(* CODESYS project HTTPSClient.library
   LanguageModelAttribute: qualified-access-only
   DefaultNamespace: HTTPS
   Description: HTTPS Client for sending http request to a webserver.
   Author: Turck Vilant Oy
   DocFormat: reStructuredText
   Title: HTTPS Client
   Version: 1.0.0.1
   Company: CODESYS GmbH
   Placeholder: HTTPSClient

Project tree, tasks and I/O mapping:
  libraries: CAA Behaviour Model, 3.5.19.0 (CAA Technical Workgroup); StringUtils, 3.5.18.0 (System); Util, 3.5.19.0 (System); Net Base Services, 3.5.19.20 (3S - Smart Software Solutions GmbH)
  HTTPRequest/
    Function Blocks/
      function block HttpsClient [ST]: StartAction, StringToURL, CyclicAction, prvResetOutputs, CreateRequest, ResetAction, prvAbort, ParseResult
    Enums/
      data type STATE
      data type REQUEST_TYPE
      data type ERROR
      data type CONTENT_TYPE
    Structs/
      data type URL
      data type HttpResult
    Functions/
      function URLDecoder [ST]
      BASE64/
        function block BASE64_DECODE [ST]
        function block BASE64_ENCODE [ST]
        function CODE [ST]
      UTF-8/
        global variables GVL_UTF8
        function ConvertUTF16toUTF8 [ST]
        function ConvertUTF8toUTF16 [ST]
        function IsLegalUTF8 [ST]
      function Concat [ST]
    Constants/
      global variables GVL
    Params/
      global variables Param
  00000000-0000-0000-0000-000000000000|C:\Users\m.lamp\Documents\license.txt
  license
*)

// HTTPRequest/Enums/STATE
// State of requests
{attribute 'qualified_only'}
{attribute 'hide'}
TYPE STATE :
(
	START := 0,
	INIT,
	REQUEST,
	RESPONSE,
	ERROR,
	IDLE
);
END_TYPE

// HTTPRequest/Enums/REQUEST_TYPE
// Types of http requests
TYPE REQUEST_TYPE :
(
	GET := 0, // http GET
	POST := 1, // http POST (needs input pwsPostValue) 
	DELETE := 2, // http DELETE
	PUT := 3, // http PUT (needs input pwsPostValue) 
	HEAD := 4 // http HEAD
);
END_TYPE

// HTTPRequest/Structs/URL
// URL structure
TYPE URL :
STRUCT
	wsProtocol	: WSTRING(5); 	// Protocol e.g. http, NOTE: ONLY HTTP IS SUPPORTED! 
	wsDomain	: WSTRING(255); 	// The domain e.g. 'twitter.api.com'
	uiPort		: UINT;			// Port of the server
	wsPath		: WSTRING(255);	// The path e.g. '/1.1/statuses/update.json'
END_STRUCT
END_TYPE

// HTTPRequest/Enums/ERROR
{attribute 'qualified_only'}
TYPE ERROR :
(
	NO_ERROR := 0, // No error
	TIME_OUT := 1, // Time out
	UNEXPECTED_ERROR := 2, // Unexpected error
	TCP_INIT_ERROR := 3, // Unable to initialize the TCP socket
	TCP_READ_ERROR := 4, // Error while reading response
	TCP_WRITE_ERROR := 5, // Error while sending the request
	MISSING_POST_VALUE := 6, // Current request type needs a post value
	RESULT_PARSE_ERROR := 7 // Error while parsing the response
);
END_TYPE

// HTTPRequest/Structs/HttpResult
// The result of a http request
TYPE HttpResult :
STRUCT
	iStatus					: INT; // http status
	wsHeader				: WSTRING(g_udiMaxHeaderSize); // http header as WSTRING
	wsContent				: WSTRING(g_udiMaxResponseSize); // The result of the request as WSTRING
	sHeader					: STRING(g_udiMaxHeaderSize); // http header as STRING
	sContent				: STRING(g_udiMaxResponseSize); // The result of the request as STRING
	diContentLength			: DINT; // Length of wsContent
END_STRUCT
END_TYPE

// HTTPRequest/Enums/CONTENT_TYPE
{attribute 'qualified_only'}
{attribute 'strict'}
TYPE CONTENT_TYPE :
(
	APPLICATION_FORM := 0, // HTML-Formulardaten an CGI 
	APPLICATION_JSON // enthält einen String in JavaScript-Objekt-Notation
);
END_TYPE

// HTTPRequest/Constants/GVL
{attribute 'hide'}
VAR_GLOBAL CONSTANT
	gc_wsBLANK : WSTRING(1) := " ";
	gc_wsLF	: WSTRING(2) :=	"$R$N";
	gc_wsDoubleLF	: WSTRING(4) :=	"$R$N$R$N";
	gc_wsContentLength	: WSTRING(15) := "Content-Length:";
	gc_wsChunked		: WSTRING(26) := "Transfer-Encoding: chunked";
	gc_wsHex	: WSTRING(3) :=	"16#";
END_VAR

// HTTPRequest/Functions/UTF-8/GVL_UTF8
{attribute 'hide'}
VAR_GLOBAL CONSTANT
	trailingBytesForUTF8 : ARRAY[0..255] OF BYTE := [
				0,0,0,0,0,0,0,0,0,0,0,0,0,0,0,0, 0,0,0,0,0,0,0,0,0,0,0,0,0,0,0,0,
				0,0,0,0,0,0,0,0,0,0,0,0,0,0,0,0, 0,0,0,0,0,0,0,0,0,0,0,0,0,0,0,0,
				0,0,0,0,0,0,0,0,0,0,0,0,0,0,0,0, 0,0,0,0,0,0,0,0,0,0,0,0,0,0,0,0,
				0,0,0,0,0,0,0,0,0,0,0,0,0,0,0,0, 0,0,0,0,0,0,0,0,0,0,0,0,0,0,0,0,
				0,0,0,0,0,0,0,0,0,0,0,0,0,0,0,0, 0,0,0,0,0,0,0,0,0,0,0,0,0,0,0,0,
				0,0,0,0,0,0,0,0,0,0,0,0,0,0,0,0, 0,0,0,0,0,0,0,0,0,0,0,0,0,0,0,0,
				1,1,1,1,1,1,1,1,1,1,1,1,1,1,1,1, 1,1,1,1,1,1,1,1,1,1,1,1,1,1,1,1,
				2,2,2,2,2,2,2,2,2,2,2,2,2,2,2,2, 3,3,3,3,3,3,3,3,4,4,4,4,5,5,5,5
			];
	firstByteMark : ARRAY[0..6] OF BYTE := [ 16#00, 16#00, 16#C0, 16#E0, 16#F0, 16#F8, 16#FC ];
	
	offsetsFromUTF8: ARRAY[0..5] OF DWORD := [ 16#00000000, 16#00003080, 16#000E2080, 
             16#03C82080, 16#FA082080, 16#82082080 ];
	
	halfShift : INT := 10; (* used FOR shifting BY 10 bits *)

	halfBase : DWORD := 16#0010000;
	halfMask : DWORD := 16#3FF;
	
	UNI_REPLACEMENT_CHAR : DWORD := 16#0000FFFD;
	
	UNI_MAX_BMP : DWORD := 16#0000FFFF;
	UNI_MAX_UTF16 : DWORD := 16#0010FFFF;
	UNI_MAX_UTF32 : DWORD := 16#7FFFFFFF;
	UNI_MAX_LEGAL_UTF32 : DWORD := 16#0010FFFF;
	
	byteMask : DWORD := 16#BF;
	byteMark : DWORD := 16#80;
	UNI_SUR_HIGH_START : DWORD := 16#D800;
 	UNI_SUR_HIGH_END : DWORD := 16#DBFF;
 	UNI_SUR_LOW_START : DWORD := 16#DC00;
 	UNI_SUR_LOW_END : DWORD := 16#DFFF;
	
	ERR_OK : UDINT := 16#0000;	(* The operation succeeded *)
	ERR_SOURCE_EXHAUSTED : UDINT := 16#40A0; (* Used for UTF8 helper *)
	ERR_TARGET_EXHAUSTED : UDINT := 16#40A1; (* Used for UTF8 helper *)
	ERR_SOURCE_ILLEGAL : UDINT := 16#40A2; (* Used for UTF8 helper *)
	
END_VAR

// HTTPRequest/Params/Param
// HTTPClient parameters
VAR_GLOBAL CONSTANT
	g_udiMaxRequestSize : UDINT := 16000; // Maximum size of the http request in btyes
	g_udiMaxResponseSize : UDINT := 16000; // Maximum size of the http response in bytes
	g_udiMaxHeaderSize : UDINT := 4000; // Maximum size of the http header in bytes
END_VAR

// HTTPRequest/Function Blocks/HttpsClient
// Functionblock to send http GET and POST requests.
//{attribute 'hide_all_locals'}
FUNCTION_BLOCK HttpsClient EXTENDS CBM.ETrigTo
VAR_INPUT
	sURL					: STRING(1024); // URL of the web server
	eRequestType			: REQUEST_TYPE := REQUEST_TYPE.GET;	// Type of the request: POST or GET
	eContentType			: CONTENT_TYPE := CONTENT_TYPE.APPLICATION_FORM; // HTTP Content-Type of the request
	pwsAdditionalHeader		: POINTER TO WSTRING; // Additional HTTP header
	pwsPostValue			: POINTER TO WSTRING; // Post parameter
	httpsTLSContext 		: NBS.ITLSContext := 0; // TLS context for HTTPS
END_VAR
VAR_OUTPUT
	eError					: ERROR; // Current error state
	httpResult				: HttpResult; // The result of the request
	_url					: URL;
	// Helpers	
	_eState 				: STATE;
END_VAR
VAR
	// TCP Connection
	_tcp_client 			: NBS.TCP_Client;
	_tcp_read 				: NBS.TCP_Read;
	_tcp_write 				: NBS.TCP_Write;
	_IPAddr 				: NBS.IPv4Address := (ipAddress := '83.150.96.4');
	_IIPAddr	 			: NBS.IIPAddress := _IPAddr;
	_resolve_host_name 		: NBS.ResolveHostname;	
	_wsRequest 				: WSTRING(g_udiMaxRequestSize);
	_abRequest 				: ARRAY[0..g_udiMaxRequestSize] OF BYTE;
	_sContent				: STRING(g_udiMaxResponseSize); 
	_pbContent				: POINTER TO BYTE;
	_wsContent				: WSTRING(g_udiMaxResponseSize);
	
	
END_VAR

SUPER^();
eError := iError;

{attribute 'hide'}
METHOD StartAction : BOOL
VAR_INPUT
END_VAR
VAR
END_VAR
END_METHOD

{attribute 'hide'}
// Converts a string to an url.
METHOD StringToURL : ERROR
VAR_INPUT
	wsUrl		: WSTRING(1024);	// The url as string
END_VAR
VAR_IN_OUT
	url			: URL; // The URL struct
END_VAR
VAR
	wsTemp		: WSTRING(1024);
	wsPort		: WSTRING(6);
	i			: INT;
END_VAR
VAR CONSTANT
	wsDel		: WSTRING(3) := "://";
	wsPortDel	: WSTRING(1) := ":";
	wsPathStart	: WSTRING(1) := "/";
END_VAR
// Find '://'
i := Stu.StrFindW(pst1 := ADR(wsUrl), pst2 := ADR(wsDel), uiSearchStart := 1);
IF i > 0 THEN
	Stu.StrMidW(pwst := ADR(wsUrl),
				uiInputBufferSize := SIZEOF(wsUrl),
				iLength := DINT_TO_INT(Stu.StrLenW(ADR(wsUrl))) - i - DINT_TO_INT(Stu.StrLenW(ADR(wsDel))) + 1,
				iPosition := i +  DINT_TO_INT(Stu.StrLenW(ADR(wsDel))),
				pwstResult := ADR(wsTemp),
				uiResultBufferSize := SIZEOF(wsTemp));
	// Set protocol			
	Stu.StrMidW(pwst := ADR(wsUrl),
				uiInputBufferSize := SIZEOF(wsUrl),
				iLength := i - 1,
				iPosition := 1,
				pwstResult := ADR(url.wsProtocol),
				uiResultBufferSize := SIZEOF(url.wsProtocol));
ELSE
	url.wsProtocol := "http";
	wsTemp := wsUrl;
END_IF

// Find path start '/'
i := Stu.StrFindW(pst1 := ADR(wsTemp), pst2 := ADR(wsPathStart), uiSearchStart := 1);
IF i > 0 THEN
	// set path
	Stu.StrMidW(pwst := ADR(wsTemp),
				uiInputBufferSize := SIZEOF(wsTemp),
				iLength := DINT_TO_INT(Stu.StrLenW(ADR(wsTemp))) - i + DINT_TO_INT(Stu.StrLenW(ADR(wsPathStart))),
				iPosition := i + DINT_TO_INT(Stu.StrLenW(ADR(wsPathStart))) - 1,
				pwstResult := ADR(url.wsPath),
				uiResultBufferSize := SIZEOF(url.wsPath));	
				
	Stu.StrMidW(pwst := ADR(wsTemp),
				uiInputBufferSize := SIZEOF(wsTemp),
				iLength := i - 1,
				iPosition := 1,
				pwstResult := ADR(wsTemp),
				uiResultBufferSize := SIZEOF(wsTemp));			
ELSE
	url.wsPath := "";
END_IF


i := Stu.StrFindW(pst1 := ADR(wsTemp), pst2 := ADR(wsPortDel), uiSearchStart := 1);
IF i > 0 THEN
	// set domain
	Stu.StrMidW(pwst := ADR(wsTemp),
				uiInputBufferSize := SIZEOF(wsTemp),
				iLength := i - 1,
				iPosition := 1,
				pwstResult := ADR(url.wsDomain),
				uiResultBufferSize := SIZEOF(url.wsDomain));	
	// set port
	Stu.StrMidW(pwst := ADR(wsTemp),
				uiInputBufferSize := SIZEOF(wsTemp),
				iLength := DINT_TO_INT(Stu.StrLenW(ADR(wsTemp)) - i - Stu.StrLenW(ADR(wsPortDel))) + 1,
				iPosition := i + DINT_TO_INT(Stu.StrLenW(ADR(wsPortDel))),
				pwstResult := ADR(wsPort),
				uiResultBufferSize := SIZEOF(wsPort));
	url.uiPort := WSTRING_TO_UINT(wsPort);				
ELSIF url.wsProtocol = "http" THEN
	url.wsDomain := wsTemp;
	url.uiPort := 80;
ELSIF url.wsProtocol = "https" THEN
	url.wsDomain := wsTemp;
	url.uiPort := 443;
ELSE
	url.wsDomain := wsTemp;
	url.uiPort := 80;
END_IF

IF url.wsPath = "" THEN
	url.wsPath := "/";
END_IF
END_METHOD

{attribute 'hide'}
METHOD CyclicAction : BOOL
VAR_INPUT
END_VAR
VAR
	uxiBytesRead : __UXINT;
	sDomain : STRING;
END_VAR

IF xExecute = TRUE AND _eState = STATE.IDLE THEN
	_eState := STATE.START;
END_IF

CASE _eState OF
	
STATE.IDLE: // Idle

STATE.START: // stopped
	// Parse url 
	_sContent := '';
	_pbContent := ADR(_sContent);
	_wsContent := "";
	httpResult.wsContent := "";
	httpResult.wsHeader := "";
	httpResult.diContentLength := 0;
	httpResult.iStatus := 0;
	iError := StringToURL(wsUrl := STRING_TO_WSTRING(sUrl), url := _url);
	IF iError <> ERROR.NO_ERROR THEN
		_eState := STATE.ERROR;		
		xError := TRUE;	
		RETURN;
	END_IF
	//_IPAddr.sAddr := WSTRING_TO_STRING(_url.wsDomain);
	_tcp_client(xEnable := FALSE);
	_tcp_read(xEnable := FALSE);
	_tcp_write(xExecute := FALSE);
	sDomain := WSTRING_TO_STRING(_url.wsDomain);
	_resolve_host_name(xExecute:=, sHostName:=sDomain , itfIPAddress:=_IIPAddr);
	_resolve_host_name.xExecute := TRUE;
	IF _resolve_host_name.xDone THEN
		_resolve_host_name.xExecute := FALSE;
		_eState := STATE.INIT;
	END_IF
	
	IF (eRequestType = REQUEST_TYPE.POST OR eRequestType = REQUEST_TYPE.PUT) AND (pwsPostValue = 0 OR Stu.StrLenW(pstData := pwsPostValue) = 0) THEN
		iError := ERROR.MISSING_POST_VALUE;
		_eState := STATE.ERROR;
	END_IF
	
STATE.INIT:	// init client
	_tcp_client(xEnable := TRUE, itfIPAddress := _IIPAddr, uiPort := _url.uiPort, itfTLSContext:=httpsTLSContext);
	IF _tcp_client.xBusy THEN//AND _tcp_client.hConnection <> CAA.gc_hINVALID THEN
		_eState := STATE.REQUEST;
	ELSIF _tcp_client.xError THEN
		iError := ERROR.TCP_INIT_ERROR;
		_eState := STATE.ERROR;
	END_IF
	
STATE.REQUEST:		// send message	
	CreateRequest(url := _url, pwsAdditionalHeader := pwsAdditionalHeader, pwsPostValue := pwsPostValue, wsOut := _wsRequest);
	ConvertUTF16toUTF8(sourceStart := ADR(_wsRequest), targetStart := ADR(_abRequest), dwTargetBufferSize := SIZEOF(_abRequest), bStrictConversion := FALSE);
	_tcp_write(xExecute := _tcp_client.xActive, itfConnection := _tcp_client.itfConnection, udiSize := DINT_TO_UDINT(Stu.StrLenA(ADR(_abRequest))), pData := ADR(_abRequest));
	IF _tcp_write.xDone THEN		// message sent, go back to idle mode
		_tcp_write(xExecute := FALSE);			
		_eState := STATE.RESPONSE;
	ELSIF _tcp_write.xError THEN
		iError := ERROR.TCP_WRITE_ERROR;
		_eState := STATE.ERROR;
	END_IF
	
STATE.RESPONSE:	// idle mode - wait for incomming message
	_tcp_read(xEnable := _tcp_client.xActive, itfConnection := _tcp_client.itfConnection, udiSize := SIZEOF(_sContent), pData := ADR(_sContent));
	IF _tcp_read.xReady THEN		
		_pbContent[uxiBytesRead] := 0;
		_tcp_read(xEnable := FALSE);		
		_eState := STATE.IDLE;
		ResetAction();
		ConvertUTF8toUTF16(sourceStart := ADR(_sContent), targetStart := ADR(_wsContent), dwTargetBufferSize := SIZEOF(_wsContent), bStrictConversion := FALSE);
		ParseResult(wsContent := _wsContent, httpResult := httpResult);
		xDone := TRUE;
	ELSIF _tcp_read.xError THEN		
		iError := ERROR.TCP_READ_ERROR;
		_eState := STATE.ERROR;		
		xError := TRUE;	
	END_IF		

STATE.ERROR:
	_sContent := '';
	_wsContent := "";
	ResetAction();
	_eState := STATE.IDLE;
	
END_CASE
END_METHOD

{attribute 'hide'}
METHOD prvResetOutputs : BOOL
VAR_INPUT
END_VAR
VAR
END_VAR
SUPER^.prvResetOutputs();
END_METHOD

// Builds a http request
{attribute 'hide'}
METHOD CreateRequest
VAR_INPUT
	url						: URL; // The URL of the webserver
	pwsAdditionalHeader		: POINTER TO WSTRING; // Additional HTTP header	
	pwsPostValue			: POINTER TO WSTRING; // Post parameter
END_VAR
VAR_IN_OUT
	wsOut					: WSTRING(g_udiMaxRequestSize);
END_VAR
VAR
	wsType				: WSTRING(6); // Type of the request: GET or POST
	wsContentLength		: WSTRING(5);
	wsHTTP_HEADER		: WSTRING(100) 	:= "Connection: close$000D$000AContent-Type: application/x-www-form-urlencoded";
END_VAR
VAR CONSTANT
	wsBlank				: WSTRING(1) 	:= " ";
	wsLF				: WSTRING(2) 	:= "$000D$000A";
	wsLF2				: WSTRING(4) 	:= "$000D$000A$000D$000A";
	wsHTTPVersion		: WSTRING(12) 	:= " HTTP/1.1";
	wsHTTPContetntLength	: WSTRING(17) 	:= "Content-Length: ";
	wsHTTPHost 			: WSTRING(9) 	:= "Host: ";
END_VAR
IF eRequestType = REQUEST_TYPE.GET THEN
	wsType := "GET";
ELSIF eRequestType = REQUEST_TYPE.DELETE THEN
	wsType := "DELETE";
ELSIF eRequestType = REQUEST_TYPE.HEAD THEN
	wsType := "HEAD";
ELSIF eRequestType = REQUEST_TYPE.PUT THEN
	wsType := "PUT";
ELSIF eRequestType = REQUEST_TYPE.POST THEN
	wsType := "POST";
ELSE
	wsType := "";
END_IF

IF eContentType = CONTENT_TYPE.APPLICATION_JSON THEN
	wsHTTP_HEADER := "Connection: keep-alive$000D$000AContent-Type: application/json";
END_IF

// POST or GET
wsOut := "";
Concat(ADR(wsType), ADR(wsOut), SIZEOF(wsOut));
Concat(ADR(wsBlank), ADR(wsOut), SIZEOF(wsOut));
Concat(ADR(url.wsPath), ADR(wsOut), SIZEOF(wsOut));
Concat(ADR(wsBlank), ADR(wsOut), SIZEOF(wsOut));
Concat(ADR(wsHTTPVersion), ADR(wsOut), SIZEOF(wsOut));
Concat(ADR(wsLF), ADR(wsOut), SIZEOF(wsOut));

// HTTP Header
Stu.StrConcatW(ADR(wsHTTP_HEADER), ADR(wsOut), DINT_TO_INT(SIZEOF(wsOut)));
Stu.StrConcatW(ADR(wsLF), ADR(wsOut), DINT_TO_INT(SIZEOF(wsOut)));
IF NOT Stu.StrIsNullOrEmptyA(pwsAdditionalHeader) THEN
	Stu.StrConcatW(pwsAdditionalHeader, ADR(wsOut), DINT_TO_INT(SIZEOF(wsOut)));
	Stu.StrConcatW(ADR(wsLF), ADR(wsOut), DINT_TO_INT(SIZEOF(wsOut)));
END_IF

// Host
Concat(ADR(wsHTTPHost), ADR(wsOut), SIZEOF(wsOut));
Concat(ADR(url.wsDomain), ADR(wsOut), SIZEOF(wsOut));
Concat(ADR(wsLF), ADR(wsOut), SIZEOF(wsOut));

IF eRequestType = REQUEST_TYPE.POST OR eRequestType = REQUEST_TYPE.PUT THEN
	Concat(ADR(wsHTTPContetntLength), ADR(wsOut), SIZEOF(wsOut));
	wsContentLength := DINT_TO_WSTRING(Stu.StrLenW(pwsPostValue));
	Concat(ADR(wsContentLength), ADR(wsOut), SIZEOF(wsOut));
END_IF
Concat(ADR(wsLF), ADR(wsOut), SIZEOF(wsOut));
Concat(ADR(wsLF), ADR(wsOut), SIZEOF(wsOut));

// Post content
IF eRequestType = REQUEST_TYPE.POST OR eRequestType = REQUEST_TYPE.PUT THEN
	Concat(pwsPostValue, ADR(wsOut), SIZEOF(wsOut));
END_IF
END_METHOD

{attribute 'hide'}
METHOD ResetAction
VAR_INPUT
END_VAR
_tcp_write(xExecute := FALSE);	
_tcp_read(xEnable := FALSE);	
_tcp_client(xEnable := FALSE);
END_METHOD

{attribute 'hide'}
METHOD prvAbort : BOOL
VAR_INPUT
END_VAR
VAR
END_VAR
ResetAction();
_eState := STATE.IDLE;
xAbortInProgress := FALSE;
END_METHOD

{attribute 'hide'}
METHOD ParseResult : ERROR
VAR_IN_OUT
	wsContent : WSTRING(g_udiMaxResponseSize);
	httpResult : HTTPResult;
END_VAR
VAR
	diTemp1 : DINT;
	diTemp2 : DINT;
	diContentStartPos : DINT;
	wsStatus : WSTRING(4);
	wsContentLength : WSTRING(20);
	wsContentLengthHex : WSTRING(20);
	xIsChunked : BOOL;
END_VAR
// Find HTTP status
diTemp1 := Stu.StrFindW(pst1 := ADR(wsContent), pst2 := ADR(gc_wsBLANK), uiSearchStart := 0);
diTemp2 := Stu.StrFindW(pst1 := ADR(wsContent), pst2 := ADR(gc_wsBLANK), uiSearchStart := DINT_TO_UINT(diTemp1 + 1));
IF diTemp1 < 1 OR diTemp2 < 1 THEN
	ParseResult := ERROR.RESULT_PARSE_ERROR;
	RETURN;
END_IF
Stu.StrMidW(	pwst := ADR(wsContent), 
				uiInputBufferSize := SIZEOF(wsContent), 
				iLength := DINT_TO_INT(diTemp2 - diTemp1), 
				iPosition := DINT_TO_INT(diTemp1), 
				pwstResult := ADR(wsStatus), 
				uiResultBufferSize := SIZEOF(wsStatus));
httpResult.iStatus := WSTRING_TO_INT(wsStatus);

// Find header
diTemp1 := Stu.StrFindW(pst1 := ADR(wsContent), pst2 := ADR(gc_wsLF), uiSearchStart := DINT_TO_UINT(diTemp2 + 1));
diTemp2 := Stu.StrFindW(pst1 := ADR(wsContent), pst2 := ADR(gc_wsDoubleLF), uiSearchStart := DINT_TO_UINT(diTemp1 + 1));
IF diTemp1 < 1 OR diTemp2 < 1 THEN
	ParseResult := ERROR.RESULT_PARSE_ERROR;
	RETURN;
END_IF
Stu.StrMidW(	pwst := ADR(wsContent), 
				uiInputBufferSize := SIZEOF(wsContent), 
				iLength := DINT_TO_INT(diTemp2 - diTemp1) - 2, 
				iPosition := DINT_TO_INT(diTemp1) + 2, 
				pwstResult := ADR(httpResult.wsHeader), 
				uiResultBufferSize := SIZEOF(httpResult.wsHeader));

diContentStartPos := diTemp2 + 4;

xIsChunked := Stu.StrFindW(pst1 := ADR(httpResult.wsHeader), pst2 := ADR(gc_wsChunked), uiSearchStart := 0) > 0;
IF xIsChunked THEN
	// Convert chunked data
	diTemp1 := diContentStartPos;
	// Get data length
	diTemp2 := Stu.StrFindW(pst1 := ADR(wsContent), pst2 := ADR(gc_wsLF), uiSearchStart := DINT_TO_UINT(diTemp1));
	IF diTemp2 < 1 THEN
		ParseResult := ERROR.RESULT_PARSE_ERROR;
		RETURN;
	END_IF
	Stu.StrMidW(	pwst := ADR(wsContent), 
					uiInputBufferSize := SIZEOF(wsContent), 
					iLength := DINT_TO_INT(diTemp2 - diTemp1), 
					iPosition := DINT_TO_INT(diTemp1), 
					pwstResult := ADR(wsContentLength), 
					uiResultBufferSize := SIZEOF(wsContentLength));
	wsContentLengthHex := gc_wsHex;
	Stu.StrConcatW(pstFrom := ADR(wsContentLength), pstTo := ADR(wsContentLengthHex), iBufferSize := SIZEOF(wsContentLengthHex));
	httpResult.diContentLength := WSTRING_TO_DINT(wsContentLengthHex);
	// Copy content
	Stu.StrMidW(	pwst := ADR(wsContent), 
					uiInputBufferSize := SIZEOF(wsContent), 
					iLength := DINT_TO_INT(httpResult.diContentLength), 
					iPosition := DINT_TO_INT(diTemp2 + 2), 
					pwstResult := ADR(httpResult.wsContent), 
					uiResultBufferSize := SIZEOF(httpResult.wsContent));
ELSE	
	// Find content
	diTemp2 := Stu.StrLenW(pstData := ADR(wsContent));
	IF diTemp2 < 0 THEN
		ParseResult := ERROR.RESULT_PARSE_ERROR;
		RETURN;
	END_IF
	Stu.StrMidW(	pwst := ADR(wsContent), 
					uiInputBufferSize := SIZEOF(wsContent), 
					iLength := DINT_TO_INT(diTemp2 - diContentStartPos + 1), 
					iPosition := DINT_TO_INT(diContentStartPos), 
					pwstResult := ADR(httpResult.wsContent), 
					uiResultBufferSize := SIZEOF(httpResult.wsContent));
	httpResult.diContentLength := diTemp2 - diContentStartPos + 1;
END_IF

// Copy WSTRING to STRING values
ConvertUTF16toUTF8(sourceStart := ADR(httpResult.wsHeader), targetStart := ADR(httpResult.sHeader), dwTargetBufferSize := SIZEOF(httpResult.sHeader), bStrictConversion := FALSE);
ConvertUTF16toUTF8(sourceStart := ADR(httpResult.wsContent), targetStart := ADR(httpResult.sContent), dwTargetBufferSize := SIZEOF(httpResult.sContent), bStrictConversion := FALSE);
END_METHOD

END_FUNCTION_BLOCK

// HTTPRequest/Functions/UTF-8/ConvertUTF16toUTF8
// Converts a WSTRING to STRING
FUNCTION ConvertUTF16toUTF8 : UDINT
VAR_INPUT
 	sourceStart : POINTER TO WORD;	// Pointer to WSTRING
	targetStart : POINTER TO BYTE;	// Pointer to STRING
	dwTargetBufferSize : DWORD;		// Size of STRING
	bStrictConversion : BOOL;
END_VAR
VAR
	source : POINTER TO WORD;
	sourceEnd : POINTER TO WORD;
	oldSource : POINTER TO WORD;
	target : POINTER TO BYTE;
	targetEnd : POINTER TO BYTE;
	ch : DWORD;
	ch2 : DWORD;
	bytesToWrite : WORD := 0;
	bytesToWriteSave : WORD := 0;
END_VAR

ConvertUTF16toUTF8 := ERR_OK;
source := sourceStart;
target := targetStart;
sourceEnd := source + Stu.StrLenW(source)*2 + 1; // Add the terminating 0
targetEnd := target + dwTargetBufferSize;
WHILE source < sourceEnd DO
	bytesToWrite := 0;
    oldSource := source; // In CASE we have TO back up because OF target overflow.
    ch := WORD_TO_DWORD(source^);
	source := source + 2;
    (* If we have a surrogate pair, convert to UTF32 first. *)
    IF (ch >= UNI_SUR_HIGH_START AND ch <= UNI_SUR_HIGH_END) THEN
        (* If the 16 bits following the high surrogate are in the source buffer... *)
        IF (source < sourceEnd) THEN
        	ch2 := WORD_TO_DWORD(source^);
        	(* If it's a low surrogate, convert to UTF32. *)
			IF (ch2 >= UNI_SUR_LOW_START AND ch2 <= UNI_SUR_LOW_END) THEN
				ch := SHL(ch - UNI_SUR_HIGH_START, halfShift) + (ch2 - UNI_SUR_LOW_START) + halfBase;
				source := source + 2;
			ELSIF (bStrictConversion) THEN
				(* it's an unpaired high surrogate *)
				source := source - 2; // return to the illegal value itself 
				ConvertUTF16toUTF8 := ERR_SOURCE_ILLEGAL;
				EXIT;
			END_IF
		ELSE 
		 	(* We don't have the 16 bits following the high surrogate. *)
			source := source - 2; // return to the high surrogate
			ConvertUTF16toUTF8 := ERR_SOURCE_EXHAUSTED;
			EXIT;
		END_IF
	ELSIF (bStrictConversion) THEN
        (* UTF-16 surrogate values are illegal in UTF-32 *)
        IF (ch >= UNI_SUR_LOW_START AND ch <= UNI_SUR_LOW_END) THEN
        	source := source - 2; // RETURN TO the illegal value itself
        	ConvertUTF16toUTF8 := ERR_SOURCE_ILLEGAL;
        	EXIT;
        END_IF
    END_IF
    (* Figure out how many bytes the result will require *)
    IF (ch < 16#80) THEN      
		bytesToWrite := 1;
    ELSIF (ch < 16#800) THEN     
		bytesToWrite := 2;
    ELSIF (ch < 16#10000) THEN   
		bytesToWrite := 3;
    ELSIF (ch < 16#110000) THEN  
		bytesToWrite := 4;
    ELSE       
		bytesToWrite := 3;
        ch := UNI_REPLACEMENT_CHAR;
    END_IF

    target := target + bytesToWrite;
    IF (target > targetEnd) THEN
        source := oldSource; // Back up source pointer! 
        target := target - bytesToWrite; 
		ConvertUTF16toUTF8 := ERR_TARGET_EXHAUSTED; 
		EXIT;
   	END_IF
	bytesToWriteSave := bytesToWrite;
    IF bytesToWrite = 4 THEN
		target := target - 1;
		target^ := DWORD_TO_BYTE((ch OR byteMark) AND byteMask); 
		ch := SHR(ch, 6);
		bytesToWrite := 3;
	END_IF
	IF bytesToWrite = 3 THEN
		target := target - 1;
		target^ := DWORD_TO_BYTE((ch OR byteMark) AND byteMask); 
		ch := SHR(ch, 6);
		bytesToWrite := 2;
	END_IF
	IF bytesToWrite = 2 THEN
		target := target - 1;
		target^ := DWORD_TO_BYTE((ch OR byteMark) AND byteMask); 
		ch := SHR(ch, 6);
		bytesToWrite := 1;
	END_IF
	IF bytesToWrite = 1 THEN
		target := target - 1;
		target^ := DWORD_TO_BYTE(ch OR firstByteMark[bytesToWriteSave]);
	END_IF
    target := target + bytesToWriteSave;
END_WHILE

END_FUNCTION

// HTTPRequest/Functions/UTF-8/ConvertUTF8toUTF16
// Converts a STRING to WSTRING.
FUNCTION ConvertUTF8toUTF16 : UDINT
VAR_INPUT
 	sourceStart : POINTER TO BYTE; 	// Pointer to STRING
	targetStart : POINTER TO WORD;	// Pointer to WSTRING
	dwTargetBufferSize : DWORD;		// Size of the WSTRING
	bStrictConversion : BOOL;
END_VAR
VAR
	source : POINTER TO BYTE;
	sourceEnd : POINTER TO BYTE;
	target : POINTER TO WORD;
	targetEnd : POINTER TO WORD;
	ch : DWORD;
	extraBytesToRead : WORD;
	extraBytesToReadSave : WORD;
END_VAR

ConvertUTF8toUTF16 := ERR_OK;
source := sourceStart;
target := targetStart;
sourceEnd := source + Stu.StrLenA(source) + 1; // Add the terminating 0 
targetEnd := target + dwTargetBufferSize;
WHILE (source < sourceEnd) DO
	ch := 0;
	extraBytesToRead := trailingBytesForUTF8[source^];
	IF (source + extraBytesToRead >= sourceEnd) THEN
		ConvertUTF8toUTF16 := ERR_SOURCE_EXHAUSTED;
		EXIT;
	END_IF
	(* Do this check whether lenient or strict *)
	IF (NOT IsLegalUTF8(source, WORD_TO_INT(extraBytesToRead+1)) AND bStrictConversion) THEN
		ConvertUTF8toUTF16 := ERR_SOURCE_ILLEGAL;
		EXIT;
	END_IF
	(*
	* The cases all fall through. See "Note A" below.
	*)
	extraBytesToReadSave := extraBytesToRead;
	IF extraBytesToRead = 5 THEN
		ch := ch + source^;
		source := source + 1;
		ch := SHL(ch, 6); (* remember, illegal UTF-8 *)
		extraBytesToRead := 4;
	END_IF
	IF extraBytesToRead = 4 THEN
		ch := ch + source^;
		source := source + 1;
		ch := SHL(ch, 6); (* remember, illegal UTF-8 *)
		extraBytesToRead := 3;
	END_IF
	IF extraBytesToRead = 3 THEN
		ch := ch + source^;
		source := source + 1;
		ch := SHL(ch, 6); 
		extraBytesToRead := 2;
	END_IF
	IF extraBytesToRead = 2 THEN
		ch := ch + source^;
		source := source + 1;
		ch := SHL(ch, 6); 
		extraBytesToRead := 1;
	END_IF
	IF extraBytesToRead = 1 THEN
		ch := ch + source^;
		source := source + 1;
		ch := SHL(ch, 6); 
		extraBytesToRead := 0;
	END_IF
	IF extraBytesToRead = 0 THEN
		ch := ch + source^;
		source := source + 1;
	END_IF
	ch := ch - offsetsFromUTF8[extraBytesToReadSave];

	IF (target >= targetEnd) THEN
		// We don't return the source yet: source -= (extraBytesToRead+1); /* Back up source POINTER! */
		ConvertUTF8toUTF16 := ERR_TARGET_EXHAUSTED; 
		EXIT;
	END_IF
	IF (ch <= UNI_MAX_BMP) THEN 
		(* Target is a character <= 0xFFFF *)
		(* UTF-16 surrogate values are illegal in UTF-32 *)
		IF (ch >= UNI_SUR_HIGH_START AND ch <= UNI_SUR_LOW_END) THEN
			IF (bStrictConversion) THEN
				ConvertUTF8toUTF16 := ERR_SOURCE_ILLEGAL;
				EXIT;
			ELSE 
				target^ := DWORD_TO_WORD(UNI_REPLACEMENT_CHAR);
				target := target + 2;
			END_IF
		ELSE
			target^ := DWORD_TO_WORD(ch); (* normal case *)
			target := target + 2;
		END_IF
	ELSIF (ch > UNI_MAX_UTF16) THEN
		IF (bStrictConversion) THEN
			ConvertUTF8toUTF16 := ERR_SOURCE_ILLEGAL;
			// We don't return the source yet: source -= (extraBytesToRead+1); (* return to the start *)
			EXIT; (* Bail out; shouldn't continue *)
		ELSE 
			target^ := DWORD_TO_WORD(UNI_REPLACEMENT_CHAR);
			target := target + 2;
		END_IF
	ELSE 
		(* target is a character in range 0xFFFF - 0x10FFFF. *)
		IF (target + 1 >= targetEnd) THEN
			// We don't return the source yet: source -= (extraBytesToRead+1); (* Back up source pointer! *)
			ConvertUTF8toUTF16 := ERR_TARGET_EXHAUSTED; 
			EXIT;
		END_IF
		ch := ch - halfBase;
		target^ := DWORD_TO_WORD(SHR(ch, halfShift) + UNI_SUR_HIGH_START);
		target := target + 2;
		target^ := DWORD_TO_WORD(ch AND halfMask + UNI_SUR_LOW_START);
		target := target + 2;
	END_IF
END_WHILE

END_FUNCTION

// HTTPRequest/Functions/UTF-8/IsLegalUTF8
{attribute 'hide'}
FUNCTION IsLegalUTF8 : BOOL
VAR_INPUT
 	source : POINTER TO BYTE;
	length : INT;
END_VAR
VAR
	a : BYTE;
	srcptr : POINTER TO BYTE;
END_VAR

IsLegalUTF8 := FALSE;
srcptr := source+length;
IF length = 4 OR length = 3 OR length = 2 OR length = 1 THEN
	IF length = 4 THEN
		srcptr := srcptr - 1;
		a := srcptr^;
		IF (a < 16#80 OR a > 16#BF) THEN
			RETURN;
		END_IF
		length := 3;
	END_IF
	IF length = 3 THEN
		srcptr := srcptr - 1;
		a := srcptr^;
		IF (a < 16#80 OR a > 16#BF) THEN
			RETURN;
		END_IF
		length := 2;
	END_IF
	IF length = 2 THEN
		srcptr := srcptr - 1;
		a := srcptr^;
		IF (a > 16#BF) THEN
			RETURN;
		END_IF
		
		CASE (source^) OF
			(* no fall-through in this inner switch *)
			16#E0: 
				IF (a < 16#A0) THEN
					RETURN; 
				END_IF
			16#ED:  
				IF (a > 16#9F) THEN
					RETURN; 
				END_IF
			16#F0:  
				IF (a < 16#90) THEN
					RETURN; 
				END_IF
			16#F4:  
				IF (a > 16#8F) THEN
					RETURN; 
				END_IF
		ELSE
			IF (a < 16#80) THEN
				RETURN;
			END_IF
		END_CASE
		length := 1;
	END_IF
	IF length = 1 THEN
		IF (source^ >= 16#80 AND source^ < 16#C2) THEN
			RETURN;
		END_IF
	END_IF
ELSE
	RETURN;
END_IF
IF (source^ > 16#F4) THEN
	RETURN;
END_IF
IsLegalUTF8 := TRUE;

END_FUNCTION

// HTTPRequest/Functions/Concat
/// This function concatenates pstFrom to pstTo if the iBufferSize from pstTo is big enough. 
/// It will return FALSE and does no concatenation if one of the strings is NULL 
/// or the buffer size is not big enough.
{attribute 'hide'}
FUNCTION Concat : BOOL
VAR_INPUT
	pstFrom : CharBufferPtr;	// simply a pointer to byte
	pstTo : CharBufferPtr;		// simply a pointer to byte
	udiBufferSize : UDINT;			// the buffer size of pstTo
END_VAR
VAR
	{attribute 'ieccodeconversion_character_array'}
	pwdFrom : POINTER TO WORD;
	{attribute 'ieccodeconversion_character_array'}
	pwdTo : POINTER TO WORD;	
	iLenFrom : DINT;
	iLenTo : DINT;
	i : DINT;
END_VAR

IF pstFrom = NULL OR pstTo = NULL THEN
	RETURN;		// return FALSE
END_IF

iLenFrom := StrLenW(pstFrom);
iLenTo := StrLenW(pstTo);

IF (iLenTo * 2) + (iLenFrom * 2) + 2 > UDINT_TO_DINT(udiBufferSize) THEN
	RETURN;		// return FALSE => result buffer not big enough
END_IF

pwdFrom := pstFrom;
pwdTo := pstTo;

// Concatenate the string pstFrom to pstTo
FOR i := 0 TO iLenFrom - 1 DO
	pwdTo[iLenTo+i] := pwdFrom[i];
END_FOR
// Set the string termination
pwdTo[iLenTo+i] := 0;
Concat := TRUE;

END_FUNCTION

// HTTPRequest/Functions/URLDecoder
// URL Decoder/Encoder (%-Encoder)
FUNCTION URLDecoder : BOOL
VAR_INPUT
	psIn	: POINTER TO STRING; // Pointer to String to decode/encode
	diSize	: DINT;				 // Size of psIn
	xEncode : BOOL;				 // TRUE -> Encode, FALSE -> DECODE
END_VAR
VAR CONSTANT
	csaChars	: ARRAY[0..35] OF STRING(3) := [ ' ',    '!',  '"',   '#',   '&',   '(',   ')',   '*',   '+',   ',',   '/',   ':',   ';',   '=',   '?',   '@',   '[',  ']',
												'%20', '%21', '%22', '%23', '%26', '%28', '%29', '%2A', '%2B', '%2C', '%2F', '%3A', '%3B', '%3D', '%3F', '%40', '%5B', '%5D'];	
END_VAR
VAR
	i, j		: UINT;
	sReplace	: STRING(3);
	sReplaceTo	: STRING(3);
	iReplacePos	: INT;
	iReplaceLength	: INT;
	iReplaceToLength	: INT;
END_VAR

IF xEncode THEN
	j := 0;
ELSE
	j := 18;
END_IF
FOR i := 0 TO 18 DO
	iReplacePos := -1;
	WHILE iReplacePos <> 0 DO
		sReplace := csaChars[i + j];
		iReplacePos := Stu.StrFindA(pst1 := psIn, pst2 := ADR(sReplace), uiSearchStart := INT_TO_UINT(iReplacePos + 1));
		IF iReplacePos > 0 THEN				
			iReplaceLength := DINT_TO_INT(Stu.StrLenA(pstData := ADR(sReplace)));
			sReplaceTo := csaChars[i + 18 - j];
			iReplaceToLength :=  DINT_TO_INT(Stu.StrLenA(pstData := ADR(sReplaceTo)));
			Stu.StrReplaceA(	pstInput := psIn, 
								uiInputBufferSize := DINT_TO_UINT(diSize),  
								pstReplaceWith := ADR(sReplaceTo), 
								iLengthInput := DINT_TO_INT(Stu.StrLenA(pstData := psIn)),
								iLengthToReplace := iReplaceLength,
								iLengthToReplaceWith := iReplaceToLength,
								iReplacePos);
		END_IF
	END_WHILE
END_FOR
URLDecoder := TRUE;
RETURN;

END_FUNCTION

// HTTPRequest/Functions/BASE64/BASE64_DECODE
// Base 64 decoder
FUNCTION_BLOCK BASE64_DECODE
VAR_INPUT
	iSizeIn : INT; // Site of 'in'
	in 		: POINTER TO WORD; // Input: Pointer to WSTRING 
	out 	: POINTER TO WORD; // Output: Pointer to WSTRING 
END_VAR
VAR_OUTPUT
	iSizeOut : INT;
END_VAR
VAR_TEMP
	a: INT;
	b: WORD;
	o: WORD;
	off: INT;
	i1: INT;
	i2: INT;
	c: INT;
	_pwsIn 	: POINTER TO WORD;
	_pwsOut 	: POINTER TO WORD;
END_VAR

IF iSizeIn <= 0 THEN iSizeOut := 0; RETURN; END_IF;
_pwsIn := in;
_pwsOut := out;
c := iSizeIn - 1;
i2 := 0;
a := 0;
b := 0;
FOR i1 := 0 TO c DO
	o := _pwsIn^;
	IF o = 61  (* = *) THEN	EXIT;
	ELSIF o > 96 (* a-z *) THEN off := 71;
	ELSIF o > 64 (* A-Z *) THEN off := 65;
	ELSIF o > 47 (* 0-9 *) THEN off := -4;
	ELSIF o = 43 (* + *) THEN off := -19;
	ELSIF o = 47 (* / *) THEN off := -16;
	END_IF;
	b := SHL(b,6) OR INT_TO_BYTE(WORD_TO_INT(o) - off);
	a := a + 6;
	IF a >= 8 THEN
		a := a - 8;
		_pwsOut^ := WORD_TO_BYTE(SHR(b,a));
		_pwsOut := _pwsOut + SIZEOF(WORD);
		i2 := i2 + 1;
		b := b AND NOT SHL(WORD#16#FFFF,a);
	END_IF;
	_pwsIn := _pwsIn + SIZEOF(WORD);
END_FOR;
iSizeOut := i2;

END_FUNCTION_BLOCK

// HTTPRequest/Functions/BASE64/BASE64_ENCODE
// Base 64 encoder
FUNCTION_BLOCK BASE64_ENCODE
VAR_INPUT
	iSizeIn : INT;
	in 		: POINTER TO WORD; // Input: Pointer to WSTRING 
	out 	: POINTER TO WORD; // Output: Pointer to WSTRING 
END_VAR
VAR_OUTPUT
	iSizeOut : INT;
END_VAR
VAR
	a: INT;
	b: WORD;
	i: INT;
	i2: INT;
	i3: INT;
	c: INT;
	BASE64: WSTRING(64) := "ABCDEFGHIJKLMNOPQRSTUVWXYZabcdefghijklmnopqrstuvwxyz0123456789+/";
	_pwsIn 	: POINTER TO WORD;
	_pwsOut 	: POINTER TO WORD;
END_VAR

IF iSizeIn <= 0 THEN
	iSizeOut := 0;
	RETURN;
END_IF;
_pwsIn := in;
_pwsOut := out;
c := iSizeIn - 1;
i2 := 0;
a := 0;
b := 0;
FOR i := 0 TO c DO
	b := SHL(b,8) OR _pwsIn^;
	a := a + 8;
	WHILE a >= 6 DO
		a := a - 6;
		_pwsOut^ := CODE(BASE64,WORD_TO_INT(SHR(b,a)) + 1);
		i2 := i2 + 1;
		_pwsOut := _pwsOut + SIZEOF(WORD);
		b := b AND NOT SHL(WORD#16#FFFF,a);
	END_WHILE;
	_pwsIn := _pwsIn + SIZEOF(WORD);
END_FOR;
IF a > 0 THEN
	_pwsOut^ := CODE(BASE64,WORD_TO_INT(SHL(b,6 - a)) + 1);
	i2 := i2 + 1;
	_pwsOut := _pwsOut + SIZEOF(WORD);
	i3 := i2 + UINT_TO_INT((NOT INT_TO_WORD(i2) AND 2#11));
	FOR i := i2 TO i3 DO
		_pwsOut^ := 61;
		_pwsOut := _pwsOut + SIZEOF(WORD);
	END_FOR;
	iSizeOut := i3 + 1;
ELSE
	iSizeOut := i2;
END_IF;

END_FUNCTION_BLOCK

// HTTPRequest/Functions/BASE64/CODE
{attribute 'hide'}
FUNCTION CODE : BYTE
VAR_INPUT
	STR : WSTRING(64);
	POS : INT;
END_VAR
VAR
	PT : POINTER TO BYTE;
END_VAR

IF pos < 1 OR pos > Stu.StrLenW(ADR(str)) THEN
	CODE := 0;
	RETURN;
ELSE
	PT := ADR(STR) + INT_TO_DWORD(pos - 1) * 2;
	CODE := pt^;
END_IF;

END_FUNCTION
